FUNCTION_BLOCK PUBLIC FB_LampOnOffAdapter EXTENDS FB_Lamp
VAR
	fbLampOnOff			: FB_LampOnOff;
END_VAR

// Reduces the control value by 5 in the range of 10 to 100.
METHOD PUBLIC DimDown
fbLampOnOff.DimDown();
IF (_ipObserver <> 0) THEN
	_ipObserver.Update(fbLampOnOff.nLightLevel);
END_IF
END_METHOD

// Increments the control value by 5 in the range of 10 to 100.
METHOD PUBLIC DimUp
fbLampOnOff.DimUp();
IF (_ipObserver <> 0) THEN
	_ipObserver.Update(fbLampOnOff.nLightLevel);
END_IF
END_METHOD

// Sets the control value to 0.
METHOD PUBLIC Off
fbLampOnOff.Off();
IF (_ipObserver <> 0) THEN
	_ipObserver.Update(fbLampOnOff.nLightLevel);
END_IF
END_METHOD

// Sets the control value to 100.
METHOD PUBLIC On
fbLampOnOff.On();
IF (_ipObserver <> 0) THEN
	_ipObserver.Update(fbLampOnOff.nLightLevel);
END_IF
END_METHOD

END_FUNCTION_BLOCK

(* stored: Version 1.1.0.1, ProductVersion 3.1.4024.12
   POU FB_LampOnOffAdapter: Id {6861e56f-4925-4d48-b460-c6a29e1d7b4e}, SpecialFunc None
   Method DimDown: Id {84e11814-c597-4c8a-ba45-dc1836b1746d}
   Method DimUp: Id {e8ed69ba-902f-4e03-b4ed-fdbdf6572586}
   Method Off: Id {f59becd6-e49e-44aa-ad75-e8c059a04953}
   Method On: Id {b40e68d0-0aa6-4e9c-8d59-67b15bde7b97} *)
